// TIA Portal V16 export
// export: Created 2021-03-04T22:04:02.8833528Z, ExportSetting WithDefaults, DisplayName Totally Integrated Automation Portal, DisplayVersion V16, DisplayName TIA Portal Version Control Interface, DisplayVersion V16, DisplayName TIA Portal Openness, DisplayVersion V16, DisplayName SINAMICS Startdrive Advanced, DisplayVersion V16, DisplayName SINAMICS Startdrive G130, G150, S120, S150, SINAMICS MV, S210, DisplayVersion V16, DisplayName SINAMICS Startdrive G110M, G120, G120C, G120D, G120P, DisplayVersion V16, DisplayName STEP 7 Professional, DisplayVersion V16, DisplayName STEP 7 Safety, DisplayVersion V16, DisplayName WinCC Professional, DisplayVersion V16
FUNCTION_BLOCK "fbErrorScroller"   // FB330, LAD
TITLE = Scrolls through the error codes for display on the HMI
{ S7_Optimized_Access := 'TRUE' }
AUTHOR : DMC
FAMILY : Error
VERSION : 0.1
// stored: AutoNumber false, IsIECCheckEnabled false, IsRetainMemResEnabled false, MemoryReserve 100, SetENOAutomatically false, UDAEnableTagReadback false
   VAR_INPUT
      bInError01 { ExternalAccessible := 'False'; ExternalVisible := 'False'; ExternalWritable := 'False'} : Bool;   // Error 1 In Error Array
      bInError02 { ExternalAccessible := 'False'; ExternalVisible := 'False'; ExternalWritable := 'False'} : Bool;   // Error 2 In Error Array
      bInError03 { ExternalAccessible := 'False'; ExternalVisible := 'False'; ExternalWritable := 'False'} : Bool;   // Error 3 In Error Array
      bInError04 { ExternalAccessible := 'False'; ExternalVisible := 'False'; ExternalWritable := 'False'} : Bool;   // Error 4 In Error Array
      bInError05 { ExternalAccessible := 'False'; ExternalVisible := 'False'; ExternalWritable := 'False'} : Bool;   // Error 5 In Error Array
      bInError06 { ExternalAccessible := 'False'; ExternalVisible := 'False'; ExternalWritable := 'False'} : Bool;   // Error 6 In Error Array
      bInError07 { ExternalAccessible := 'False'; ExternalVisible := 'False'; ExternalWritable := 'False'} : Bool;   // Error 7 In Error Array
      bInError08 { ExternalAccessible := 'False'; ExternalVisible := 'False'; ExternalWritable := 'False'} : Bool;   // Error 8 In Error Array
      bInError09 { ExternalAccessible := 'False'; ExternalVisible := 'False'; ExternalWritable := 'False'} : Bool;   // Error 9 In Error Array
      bInError10 { ExternalAccessible := 'False'; ExternalVisible := 'False'; ExternalWritable := 'False'} : Bool;   // Error 10 In Error Array
      bInError11 { ExternalAccessible := 'False'; ExternalVisible := 'False'; ExternalWritable := 'False'} : Bool;   // Error 11 In Error Array
      bInError12 { ExternalAccessible := 'False'; ExternalVisible := 'False'; ExternalWritable := 'False'} : Bool;   // Error 12 In Error Array
      bInError13 { ExternalAccessible := 'False'; ExternalVisible := 'False'; ExternalWritable := 'False'} : Bool;   // Error 13 In Error Array
      bInError14 { ExternalAccessible := 'False'; ExternalVisible := 'False'; ExternalWritable := 'False'} : Bool;   // Error 14 In Error Array
      bInError15 { ExternalAccessible := 'False'; ExternalVisible := 'False'; ExternalWritable := 'False'} : Bool;   // Error 15 In Error Array
      bInError16 { ExternalAccessible := 'False'; ExternalVisible := 'False'; ExternalWritable := 'False'} : Bool;   // Error 16 In Error Array
      bInError17 { ExternalAccessible := 'False'; ExternalVisible := 'False'; ExternalWritable := 'False'} : Bool;   // Error 17 In Error Array
      bInError18 { ExternalAccessible := 'False'; ExternalVisible := 'False'; ExternalWritable := 'False'} : Bool;   // Error 18 In Error Array
      bInError19 { ExternalAccessible := 'False'; ExternalVisible := 'False'; ExternalWritable := 'False'} : Bool;   // Error 19 In Error Array
      bInError20 { ExternalAccessible := 'False'; ExternalVisible := 'False'; ExternalWritable := 'False'} : Bool;   // Error 20 In Error Array
      bInError21 { ExternalAccessible := 'False'; ExternalVisible := 'False'; ExternalWritable := 'False'} : Bool;   // Error 21 In Error Array
      bInError22 { ExternalAccessible := 'False'; ExternalVisible := 'False'; ExternalWritable := 'False'} : Bool;   // Error 22 In Error Array
      bInError23 { ExternalAccessible := 'False'; ExternalVisible := 'False'; ExternalWritable := 'False'} : Bool;   // Error 23 In Error Array
      bInError24 { ExternalAccessible := 'False'; ExternalVisible := 'False'; ExternalWritable := 'False'} : Bool;   // Error 24 In Error Array
      bInError25 { ExternalAccessible := 'False'; ExternalVisible := 'False'; ExternalWritable := 'False'} : Bool;   // Error 25 In Error Array
      bInError26 { ExternalAccessible := 'False'; ExternalVisible := 'False'; ExternalWritable := 'False'} : Bool;   // Error 26 In Error Array
      bInError27 { ExternalAccessible := 'False'; ExternalVisible := 'False'; ExternalWritable := 'False'} : Bool;   // Error 27 In Error Array
      bInError28 { ExternalAccessible := 'False'; ExternalVisible := 'False'; ExternalWritable := 'False'} : Bool;   // Error 28 In Error Array
      bInError29 { ExternalAccessible := 'False'; ExternalVisible := 'False'; ExternalWritable := 'False'} : Bool;   // Error 29 In Error Array
      bInError30 { ExternalAccessible := 'False'; ExternalVisible := 'False'; ExternalWritable := 'False'} : Bool;   // Error 30 In Error Array
   END_VAR
   VAR_OUTPUT
      bOutErrorExists { ExternalAccessible := 'False'; ExternalVisible := 'False'; ExternalWritable := 'False'} : Bool;   // An Error Exists
      iOutScrollingErrorNumber { ExternalAccessible := 'False'; ExternalVisible := 'False'; ExternalWritable := 'False'} : Int;   // Current Index when scrolling through errors
   END_VAR
   VAR
      TON_ErrorDelay { ExternalAccessible := 'False'; ExternalVisible := 'False'; ExternalWritable := 'False'; S7_SetPoint := 'True'} : TON_TIME;   // Delay between each scroll for a new error
   END_VAR
   VAR DB_SPECIFIC
      abErrors { ExternalAccessible := 'False'; ExternalVisible := 'False'; ExternalWritable := 'False'} : Array[#ciIndexLow..#ciIndexHigh] of Bool;
   END_VAR
   VAR
      iNextScrollNum { ExternalAccessible := 'False'; ExternalVisible := 'False'; ExternalWritable := 'False'} : Int := 1;   // Index of next error position
      iErrorsScrollNum { ExternalAccessible := 'False'; ExternalVisible := 'False'; ExternalWritable := 'False'} : Int := 1;   // Index of current error position
      bScrolling { ExternalAccessible := 'False'; ExternalVisible := 'False'; ExternalWritable := 'False'} : Bool;   // Indicates we are scrolling
      bTON_ErrorDelay { ExternalAccessible := 'False'; ExternalVisible := 'False'; ExternalWritable := 'False'} : Bool;
   END_VAR
   VAR_TEMP
      bErrorExists : Bool;   // Error Exists
   END_VAR
   VAR CONSTANT
      ciNoErrrors : Int := 0;
      ciIndexLow : Int := 1;
      ciIndexHigh : Int := 30;
   END_VAR
   VAR_TEMP   // added for the SCL form of the ladder/FBD networks
      _w1 : Bool;
   END_VAR
BEGIN

REGION Network 1: Check for valid array indexes
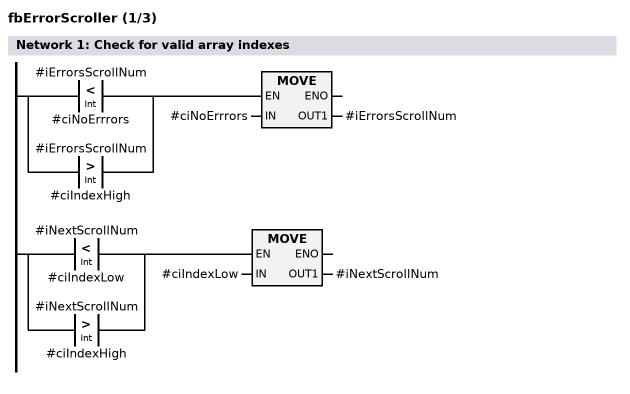
   RUNG wire#powerrail
      { S7_Templates := "SrcType := Int" } LT_Contact(in1 := #iErrorsScrollNum, in2 := #ciNoErrrors)
      wire#w1
      Move(in := #ciNoErrrors, out1 => #iErrorsScrollNum)
   END_RUNG
   RUNG wire#powerrail
      { S7_Templates := "SrcType := Int" } GT_Contact(in1 := #iErrorsScrollNum, in2 := #ciIndexHigh)
   END_RUNG wire#w1
   RUNG wire#powerrail
      { S7_Templates := "SrcType := Int" } LT_Contact(in1 := #iNextScrollNum, in2 := #ciIndexLow)
      wire#w2
      Move(in := #ciIndexLow, out1 => #iNextScrollNum)
   END_RUNG
   RUNG wire#powerrail
      { S7_Templates := "SrcType := Int" } GT_Contact(in1 := #iNextScrollNum, in2 := #ciIndexHigh)
   END_RUNG wire#w2
   // the same network as SCL:
   IF (#iErrorsScrollNum < #ciNoErrrors) OR (#iErrorsScrollNum > #ciIndexHigh) THEN
       #iErrorsScrollNum := #ciNoErrrors;
   END_IF;
   IF (#iNextScrollNum < #ciIndexLow) OR (#iNextScrollNum > #ciIndexHigh) THEN
       #iNextScrollNum := #ciIndexLow;
   END_IF;
END_REGION

REGION Network 2: Check if error exists
   // OR all of the possible errors. If any error Exists, SET bErrorExists
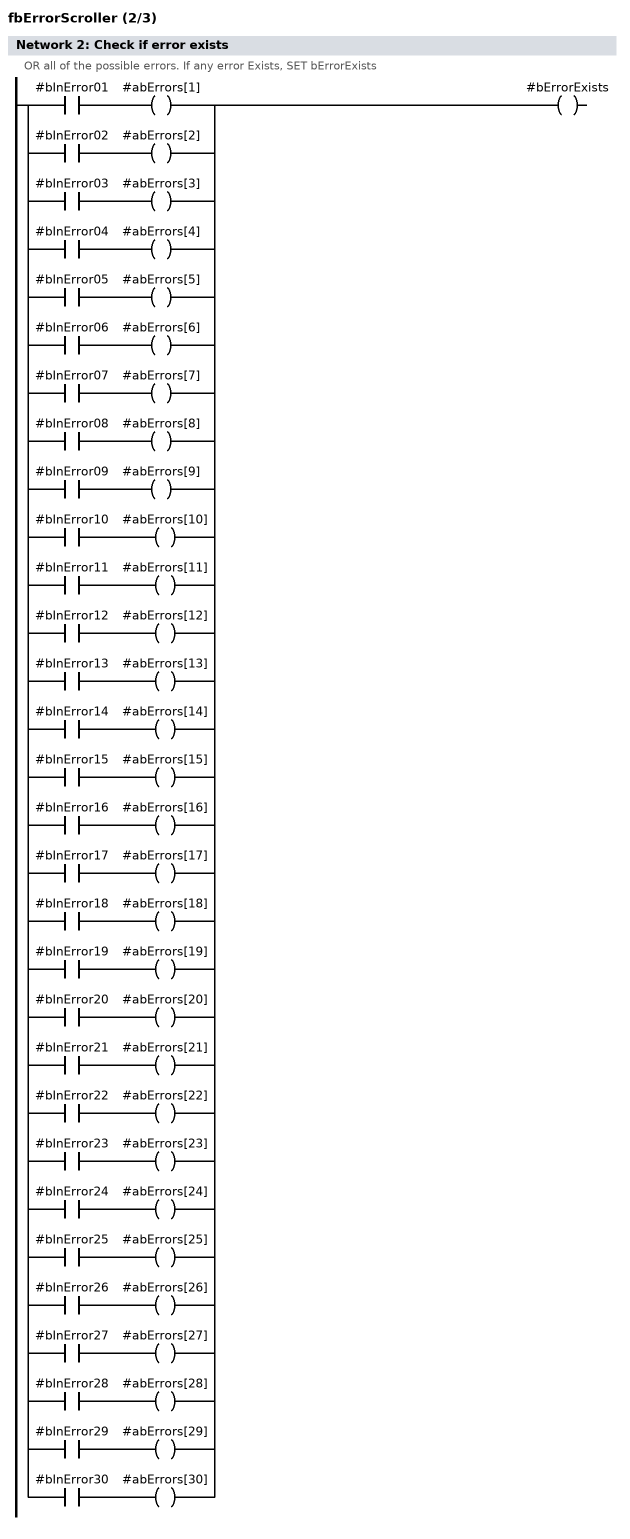
   RUNG wire#powerrail
      Contact( #bInError01 )
      Coil( #abErrors[1] )
      wire#w1
      Coil( #bErrorExists )
   END_RUNG
   RUNG wire#powerrail
      Contact( #bInError02 )
      Coil( #abErrors[2] )
   END_RUNG wire#w1
   RUNG wire#powerrail
      Contact( #bInError03 )
      Coil( #abErrors[3] )
   END_RUNG wire#w1
   RUNG wire#powerrail
      Contact( #bInError04 )
      Coil( #abErrors[4] )
   END_RUNG wire#w1
   RUNG wire#powerrail
      Contact( #bInError05 )
      Coil( #abErrors[5] )
   END_RUNG wire#w1
   RUNG wire#powerrail
      Contact( #bInError06 )
      Coil( #abErrors[6] )
   END_RUNG wire#w1
   RUNG wire#powerrail
      Contact( #bInError07 )
      Coil( #abErrors[7] )
   END_RUNG wire#w1
   RUNG wire#powerrail
      Contact( #bInError08 )
      Coil( #abErrors[8] )
   END_RUNG wire#w1
   RUNG wire#powerrail
      Contact( #bInError09 )
      Coil( #abErrors[9] )
   END_RUNG wire#w1
   RUNG wire#powerrail
      Contact( #bInError10 )
      Coil( #abErrors[10] )
   END_RUNG wire#w1
   RUNG wire#powerrail
      Contact( #bInError11 )
      Coil( #abErrors[11] )
   END_RUNG wire#w1
   RUNG wire#powerrail
      Contact( #bInError12 )
      Coil( #abErrors[12] )
   END_RUNG wire#w1
   RUNG wire#powerrail
      Contact( #bInError13 )
      Coil( #abErrors[13] )
   END_RUNG wire#w1
   RUNG wire#powerrail
      Contact( #bInError14 )
      Coil( #abErrors[14] )
   END_RUNG wire#w1
   RUNG wire#powerrail
      Contact( #bInError15 )
      Coil( #abErrors[15] )
   END_RUNG wire#w1
   RUNG wire#powerrail
      Contact( #bInError16 )
      Coil( #abErrors[16] )
   END_RUNG wire#w1
   RUNG wire#powerrail
      Contact( #bInError17 )
      Coil( #abErrors[17] )
   END_RUNG wire#w1
   RUNG wire#powerrail
      Contact( #bInError18 )
      Coil( #abErrors[18] )
   END_RUNG wire#w1
   RUNG wire#powerrail
      Contact( #bInError19 )
      Coil( #abErrors[19] )
   END_RUNG wire#w1
   RUNG wire#powerrail
      Contact( #bInError20 )
      Coil( #abErrors[20] )
   END_RUNG wire#w1
   RUNG wire#powerrail
      Contact( #bInError21 )
      Coil( #abErrors[21] )
   END_RUNG wire#w1
   RUNG wire#powerrail
      Contact( #bInError22 )
      Coil( #abErrors[22] )
   END_RUNG wire#w1
   RUNG wire#powerrail
      Contact( #bInError23 )
      Coil( #abErrors[23] )
   END_RUNG wire#w1
   RUNG wire#powerrail
      Contact( #bInError24 )
      Coil( #abErrors[24] )
   END_RUNG wire#w1
   RUNG wire#powerrail
      Contact( #bInError25 )
      Coil( #abErrors[25] )
   END_RUNG wire#w1
   RUNG wire#powerrail
      Contact( #bInError26 )
      Coil( #abErrors[26] )
   END_RUNG wire#w1
   RUNG wire#powerrail
      Contact( #bInError27 )
      Coil( #abErrors[27] )
   END_RUNG wire#w1
   RUNG wire#powerrail
      Contact( #bInError28 )
      Coil( #abErrors[28] )
   END_RUNG wire#w1
   RUNG wire#powerrail
      Contact( #bInError29 )
      Coil( #abErrors[29] )
   END_RUNG wire#w1
   RUNG wire#powerrail
      Contact( #bInError30 )
      Coil( #abErrors[30] )
   END_RUNG wire#w1
   // the same network as SCL:
   #abErrors[1] := #bInError01;
   #abErrors[2] := #bInError02;
   #abErrors[3] := #bInError03;
   #abErrors[4] := #bInError04;
   #abErrors[5] := #bInError05;
   #abErrors[6] := #bInError06;
   #abErrors[7] := #bInError07;
   #abErrors[8] := #bInError08;
   #abErrors[9] := #bInError09;
   #abErrors[10] := #bInError10;
   #abErrors[11] := #bInError11;
   #abErrors[12] := #bInError12;
   #abErrors[13] := #bInError13;
   #abErrors[14] := #bInError14;
   #abErrors[15] := #bInError15;
   #abErrors[16] := #bInError16;
   #abErrors[17] := #bInError17;
   #abErrors[18] := #bInError18;
   #abErrors[19] := #bInError19;
   #abErrors[20] := #bInError20;
   #abErrors[21] := #bInError21;
   #abErrors[22] := #bInError22;
   #abErrors[23] := #bInError23;
   #abErrors[24] := #bInError24;
   #abErrors[25] := #bInError25;
   #abErrors[26] := #bInError26;
   #abErrors[27] := #bInError27;
   #abErrors[28] := #bInError28;
   #abErrors[29] := #bInError29;
   #abErrors[30] := #bInError30;
   #bErrorExists := #bInError01 OR #bInError02 OR #bInError03 OR #bInError04 OR #bInError05 OR #bInError06 OR #bInError07 OR #bInError08 OR #bInError09 OR #bInError10 OR #bInError11 OR #bInError12 OR #bInError13 OR #bInError14 OR #bInError15 OR #bInError16 OR #bInError17 OR #bInError18 OR #bInError19 OR #bInError20 OR #bInError21 OR #bInError22 OR #bInError23 OR #bInError24 OR #bInError25 OR #bInError26 OR #bInError27 OR #bInError28 OR #bInError29 OR #bInError30;
END_REGION

REGION Network 3: Timer to change displayed error
   // ============================ Scroll errors on HMI ========================
   // Timed delay
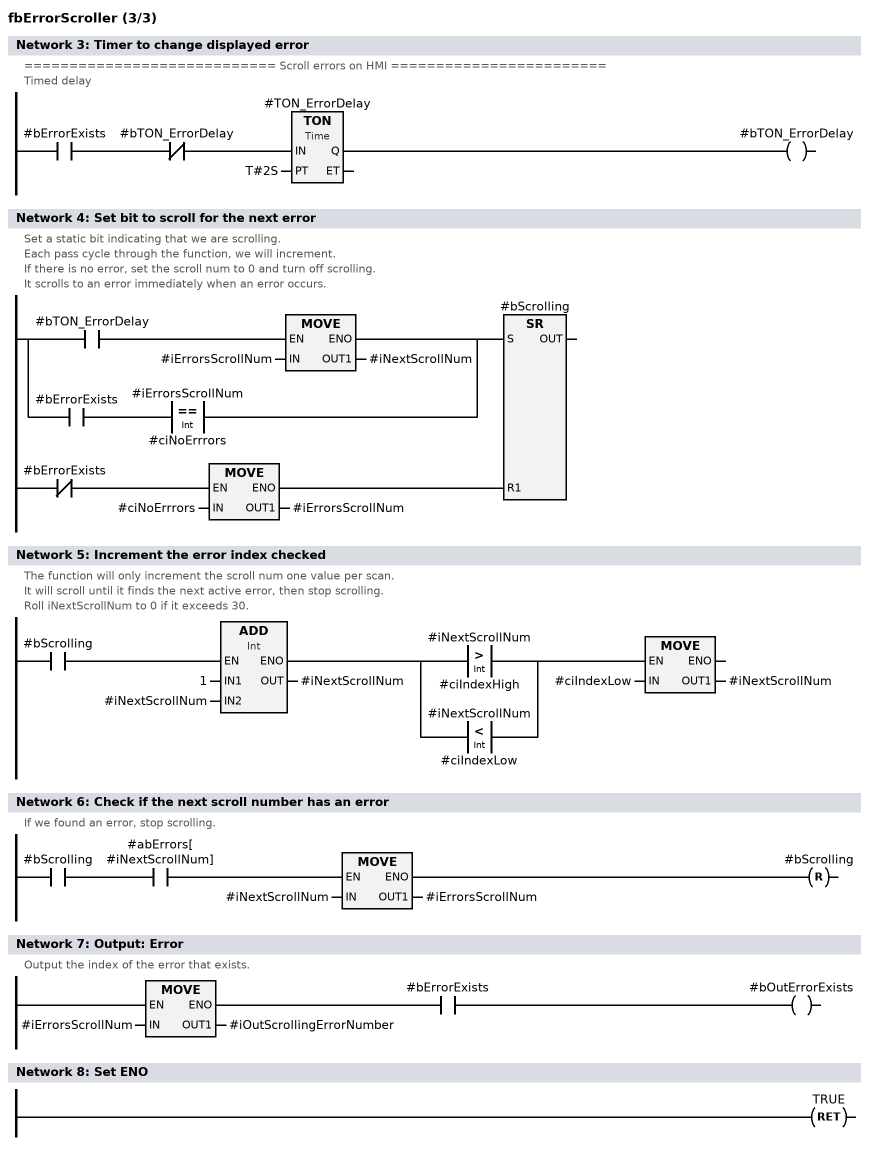
   RUNG wire#powerrail
      Contact( #bErrorExists )
      I_Contact( #bTON_ErrorDelay )
      { S7_Templates := "time_type := Time" } #TON_ErrorDelay.TON(pt := T#2S, et =>)
      Coil( #bTON_ErrorDelay )
   END_RUNG
   // the same network as SCL:
   #TON_ErrorDelay(IN := #bErrorExists AND NOT #bTON_ErrorDelay, PT := T#2S);   // TON
   #bTON_ErrorDelay := #TON_ErrorDelay.Q;
END_REGION

REGION Network 4: Set bit to scroll for the next error
   // Set a static bit indicating that we are scrolling.  
   // Each pass cycle through the function, we will increment.  
   // If there is no error, set the scroll num to 0 and turn off scrolling.  
   // It scrolls to an error immediately when an error occurs.
   RUNG wire#powerrail
      Contact( #bTON_ErrorDelay )
      { S7_GenerateENO := "TRUE" } Move(in := #iErrorsScrollNum, out1 => #iNextScrollNum)
      wire#w1
      S_SR(operand := #bScrolling, r1 := wire#w2)
   END_RUNG
   RUNG wire#powerrail
      Contact( #bErrorExists )
      { S7_Templates := "SrcType := Int" } EQ_Contact(in1 := #iErrorsScrollNum, in2 := #ciNoErrrors)
   END_RUNG wire#w1
   RUNG wire#powerrail
      I_Contact( #bErrorExists )
      { S7_GenerateENO := "TRUE" } Move(in := #ciNoErrrors, out1 => #iErrorsScrollNum)
   END_RUNG wire#w2
   // the same network as SCL:
   // ENO of a box is taken as its EN; it also drops when the box reports an error
   IF #bTON_ErrorDelay THEN #iNextScrollNum := #iErrorsScrollNum; END_IF;
   #_w1 := #bTON_ErrorDelay OR (#bErrorExists AND (#iErrorsScrollNum = #ciNoErrrors));
   IF NOT #bErrorExists THEN #iErrorsScrollNum := #ciNoErrrors; END_IF;
   IF #_w1 THEN
       #bScrolling := TRUE;   // SR flip-flop
   END_IF;
   IF NOT #bErrorExists THEN #bScrolling := FALSE; END_IF;
END_REGION

REGION Network 5: Increment the error index checked
   // The function will only increment the scroll num one value per scan.  
   // It will scroll until it finds the next active error, then stop scrolling.  
   // Roll iNextScrollNum to 0 if it exceeds 30.
   RUNG wire#powerrail
      Contact( #bScrolling )
      { S7_Templates := "SrcType := Int"; S7_GenerateENO := "TRUE" } Add(in1 := 1, in2 := #iNextScrollNum, out => #iNextScrollNum)
      wire#w1
      { S7_Templates := "SrcType := Int" } GT_Contact(in1 := #iNextScrollNum, in2 := #ciIndexHigh)
      wire#w2
      { S7_GenerateENO := "TRUE" } Move(in := #ciIndexLow, out1 => #iNextScrollNum)
   END_RUNG
   RUNG wire#w1
      { S7_Templates := "SrcType := Int" } LT_Contact(in1 := #iNextScrollNum, in2 := #ciIndexLow)
   END_RUNG wire#w2
   // the same network as SCL:
   // ENO of a box is taken as its EN; it also drops when the box reports an error
   IF #bScrolling THEN #iNextScrollNum := 1 + #iNextScrollNum; END_IF;
   IF #bScrolling AND ((#iNextScrollNum > #ciIndexHigh) OR (#iNextScrollNum < #ciIndexLow)) THEN
       #iNextScrollNum := #ciIndexLow;
   END_IF;
END_REGION

REGION Network 6: Check if the next scroll number has an error
   // If we found an error, stop scrolling.
   RUNG wire#powerrail
      Contact( #bScrolling )
      Contact( #abErrors[#iNextScrollNum] )
      { S7_GenerateENO := "TRUE" } Move(in := #iNextScrollNum, out1 => #iErrorsScrollNum)
      R_Coil( #bScrolling )
   END_RUNG
   // the same network as SCL:
   // ENO of a box is taken as its EN; it also drops when the box reports an error
   IF #bScrolling AND #abErrors[#iNextScrollNum] THEN
       #iErrorsScrollNum := #iNextScrollNum;
       #bScrolling := FALSE;
   END_IF;
END_REGION

REGION Network 7: Output: Error
   // Output the index of the error that exists.
   RUNG wire#powerrail
      { S7_GenerateENO := "TRUE" } Move(in := #iErrorsScrollNum, out1 => #iOutScrollingErrorNumber)
      Contact( #bErrorExists )
      Coil( #bOutErrorExists )
   END_RUNG
   // the same network as SCL:
   // ENO of a box is taken as its EN; it also drops when the box reports an error
   #iOutScrollingErrorNumber := #iErrorsScrollNum;
   #bOutErrorExists := #bErrorExists;
END_REGION

REGION Network 8: Set ENO
   RUNG wire#powerrail
      ReturnCoil( TRUE )
   END_RUNG
   // the same network as SCL:
   ENO := TRUE;
   RETURN;
END_REGION
END_FUNCTION_BLOCK
